// TIA Portal V17 export
// export: Created 2023-12-22T15:05:28.6198441Z, ExportSetting WithDefaults, DisplayName Totally Integrated Automation Portal, DisplayVersion V17, DisplayName TIA Portal Openness, DisplayVersion V17, DisplayName TIA Portal Version Control Interface, DisplayVersion V17, DisplayName STEP 7 Professional, DisplayVersion V17, DisplayName STEP 7 Safety, DisplayVersion V17, DisplayName WinCC Advanced, DisplayVersion V17
FUNCTION_BLOCK "Valves"   // FB250, LAD
TITLE = Клапана
{ S7_Optimized_Access := 'FALSE' }
VERSION : 0.1
// FB_Alarm - аварийный сигнал для отключения клапана (например по давлению воздуха), 0 - авария, 1 - норма
// FB_QF - сигнал готовности к работе (например, по наличию 24в в линии управления пневмораспределителем), 0 - авария, 1 - норма
// FB_Open - обратная связь датчика открытия клапана, 0 - закрыт, 1 - открыт
// FB_Close - обратная связь датчика закрытия клапана, 1 - закрыт, 0 - открыт
// Value - управление аналоговым клапаном с позиционированием, формат Real, передаётся в блок AO_ex для конвертации в выходной сигнал контроллера (PQW), для использования установите #CMD.Analog в True
// 
// Q -  постоянный сигнал управления клапаном, 0 - закрыть, 1 - открыть
// stored: AutoNumber false, IsIECCheckEnabled false, SetENOAutomatically false, UDAEnableTagReadback false
   VAR DB_SPECIFIC
      Time_DTL { S7_SetPoint := 'True'} : DTL;
   END_VAR
   VAR_TEMP   // added for the SCL form of the ladder/FBD networks
      _w1 : Bool;
   END_VAR
BEGIN

REGION Network 1: Задвижки
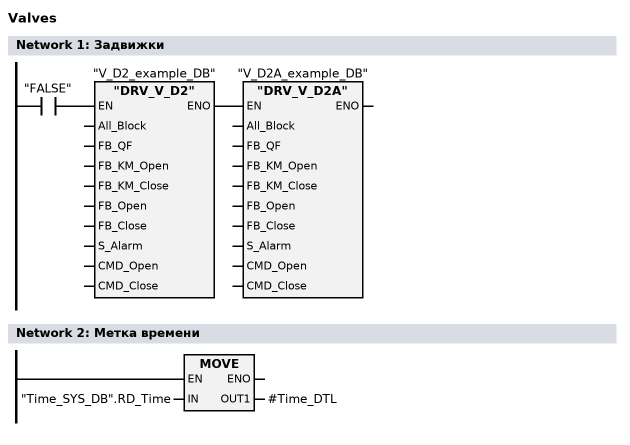
   RUNG wire#powerrail
      Contact( "FALSE" )
      "V_D2_example_DB"(All_Block :=, FB_QF :=, FB_KM_Open :=, FB_KM_Close :=, FB_Open :=, FB_Close :=, S_Alarm :=, CMD_Open :=, CMD_Close :=)
      "V_D2A_example_DB"(All_Block :=, FB_QF :=, FB_KM_Open :=, FB_KM_Close :=, FB_Open :=, FB_Close :=, S_Alarm :=, CMD_Open :=, CMD_Close :=)
   END_RUNG
   // the same network as SCL:
   "V_D2_example_DB"(EN := "FALSE", ENO => #_w1);   // "DRV_V_D2"
   IF #_w1 THEN
       "V_D2A_example_DB"();   // "DRV_V_D2A"
   END_IF;
END_REGION

REGION Network 2: Метка времени
   RUNG wire#powerrail
      Move(in := "Time_SYS_DB".RD_Time, out1 => #Time_DTL)
   END_RUNG
   // the same network as SCL:
   #Time_DTL := "Time_SYS_DB".RD_Time;
END_REGION
END_FUNCTION_BLOCK
